(* CoDeSys 2.3 library: TcMath.lib *)
(* Libraries: TcBaseMath.lib 27.7.04 12:07:55 *)

(* POU F_GetVersionTcMath, ST *)
FUNCTION F_GetVersionTcMath : 	UINT	(*Gets the library version info *)
VAR_INPUT
	nVersionElement				:	INT;
END_VAR
(*
	Possible nVersionElement parameter:
	1	:	major number
	2	:	minor number
	3	:	revision number
*)
VAR
END_VAR
(* Version history:
Date          | Version    | created under      	| Author          | Remark 
---------------------------------------------------------------------------------------- 
06/02/2004    	| 1.0.0      	| V2.9.0 (Build 959) 	| Marc S.     	| first release 
09/30/2004    	| 1.0.1      	| V2.9.0 (Build 1004)	| Marc S.     	| MODABS interface changed
09/30/2004    	| 1.0.1      	| V2.9.0 (Build 1004)	| Marc S.     	| F_GetVersionTcMath added
*) 
CASE nVersionElement OF
1:	(* major number *)
	F_GetVersionTcMath := 1;
2:	(* minor number *)
	F_GetVersionTcMath := 0;
3:	(* revision number *)
	F_GetVersionTcMath := 1;
ELSE
	F_GetVersionTcMath := 16#FFFF;
END_CASE
END_FUNCTION

(* POU FLOOR, ST *)
FUNCTION FLOOR : 	LREAL
VAR_INPUT
	lr_in	:	LREAL;
END_VAR
VAR
END_VAR
FLOOR := FW_Floor( lr_in );
END_FUNCTION

(* POU FRAC, ST *)
FUNCTION FRAC : 	LREAL
VAR_INPUT
	lr_in	:	LREAL;
END_VAR
VAR
END_VAR
FRAC := FW_LrealFrac( lr_in );
END_FUNCTION

(* POU LMOD, ST *)
FUNCTION LMOD : LREAL
VAR_INPUT
	lr_Value : LREAL;
	lr_Arg : LREAL;
END_VAR
VAR
END_VAR
IF lr_Arg = 0.0 THEN
	LMOD := LREAL#0.0;
	RETURN;
END_IF;

LMOD := lr_Value - (lr_Arg * LTRUNC(lr_Value/lr_Arg));
END_FUNCTION

(* POU LTRUNC, ST *)
FUNCTION LTRUNC : 	LREAL
VAR_INPUT
	lr_in	:	LREAL;
END_VAR
VAR
END_VAR
LTRUNC := FW_LrealTrunc( lr_in );
END_FUNCTION

(* POU MODABS, ST *)
FUNCTION MODABS : 	LREAL
VAR_INPUT
	lr_Value	:	LREAL;
	lr_Arg	: LREAL;
END_VAR
VAR
END_VAR
MODABS := FW_LrealModP( lr_Value, lr_Arg );
END_FUNCTION

(* POU MODTURNS, ST *)
FUNCTION MODTURNS : DINT
VAR_INPUT
	lr_Value : LREAL;
	lr_Arg : LREAL;
END_VAR
VAR
	lr_Tmp : LREAL;
END_VAR
IF lr_Arg = 0.0 THEN
	MODTURNS := 0;
	RETURN;
END_IF;

lr_Tmp := FLOOR(lr_Value/lr_Arg);
MODTURNS := LREAL_TO_DINT(lr_Tmp);
END_FUNCTION
